TYPE E_TrackNum :
{attribute 'qualified_only'}
{attribute 'strict'}
	(
	MainStart 	:= 1,	
	Big 		:= 2,
	Small 		:= 4,
	MainEnd		:= 3);	
END_TYPE

(* stored: Version 1.1.0.1, ProductVersion 3.1.4026.8
   DUT E_TrackNum: Id {24d8462e-8802-42e1-a024-ae520f046af2} *)
